INTERFACE ITF_RecipePoint

PROPERTY XPoint : LREAL
GET
END_GET
SET
END_SET
END_PROPERTY

PROPERTY YPoint : LREAL
GET
END_GET
SET
END_SET
END_PROPERTY

PROPERTY ZPoint : LREAL
GET
END_GET
SET
END_SET
END_PROPERTY

END_INTERFACE

(* stored: Version 1.1.0.1, ProductVersion 3.1.4024.12
   Itf ITF_RecipePoint: Id {1866ebbc-50c5-4461-ad2a-153ef9874a5f}
   Property XPoint: Id {700da9f2-6fc1-48a6-90d7-eea346a5254e}
   Get Get: Id {85550aac-052d-4724-97d4-844878d5df24}
   Set Set: Id {fc48860d-0e30-4910-a19a-bff95f055aad}
   Property YPoint: Id {5b4c59bc-56cc-4bba-acfd-7719c7e1cfd9}
   Get Get: Id {7b31a356-ad3f-4257-963a-7183f9b79d83}
   Set Set: Id {3c20c273-5fee-4866-96f6-79b15d7ac46e}
   Property ZPoint: Id {0b447f40-a7fd-4596-aebd-d873c3c8a94a}
   Get Get: Id {86f9edb5-bd54-4a3e-966a-9eef22b70afe}
   Set Set: Id {77e01db1-650d-40da-a21e-30e4dec3916d} *)
